// TIA Portal V20 export
FUNCTION "取芯伺服" : Void   // FC2, LAD
{ S7_Optimized_Access := 'TRUE' }
// stored: SetENOAutomatically false
BEGIN

REGION Network 1 (SCL)
   "取芯V90控制字".%X0 := "G2_下载".位9;
   "取芯V90控制字".%X1 := "G2_下载".位10;
   "取芯V90控制字".%X2 := "G2_下载".位11;
   "取芯V90控制字".%X3 := "G2_下载".位12;
   "取芯V90控制字".%X4 := "G2_下载".位13;
   "取芯V90控制字".%X5 := "G2_下载".位14;
   "取芯V90控制字".%X6 := "G2_下载".位15;
   "取芯V90控制字".%X7 := "G2_下载".位16;

   "取_回原模式" := "G2_下载".整型2;

   "取_绝对位置" := "G2_下载".浮点数6;
   "取_绝对速度" := "G2_下载".浮点数7;
   "取_相对位置" := "G2_下载".浮点数8;
   "取_相对位置" := "G2_下载".浮点数9;
   "取_点动速度" := "G2_下载".浮点数10;
END_REGION

REGION Network 2
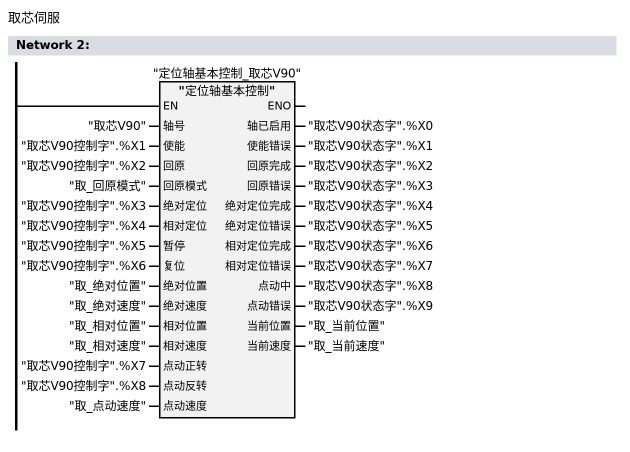
   RUNG wire#powerrail
      "定位轴基本控制_取芯V90"(轴号 := "取芯V90", 使能 := "取芯V90控制字".%X1, 回原 := "取芯V90控制字".%X2, 回原模式 := "取_回原模式", 绝对定位 := "取芯V90控制字".%X3, 相对定位 := "取芯V90控制字".%X4, 暂停 := "取芯V90控制字".%X5, 复位 := "取芯V90控制字".%X6, 绝对位置 := "取_绝对位置", 绝对速度 := "取_绝对速度", 相对位置 := "取_相对位置", 相对速度 := "取_相对速度", 点动正转 := "取芯V90控制字".%X7, 点动反转 := "取芯V90控制字".%X8, 点动速度 := "取_点动速度", 轴已启用 => "取芯V90状态字".%X0, 使能错误 => "取芯V90状态字".%X1, 回原完成 => "取芯V90状态字".%X2, 回原错误 => "取芯V90状态字".%X3, 绝对定位完成 => "取芯V90状态字".%X4, 绝对定位错误 => "取芯V90状态字".%X5, 相对定位完成 => "取芯V90状态字".%X6, 相对定位错误 => "取芯V90状态字".%X7, 点动中 => "取芯V90状态字".%X8, 点动错误 => "取芯V90状态字".%X9, 当前位置 => "取_当前位置", 当前速度 => "取_当前速度")
   END_RUNG
   // the same network as SCL:
   "定位轴基本控制_取芯V90"(轴号 := "取芯V90",   // "定位轴基本控制"
                   使能 := "取芯V90控制字".%X1,
                   回原 := "取芯V90控制字".%X2,
                   回原模式 := "取_回原模式",
                   绝对定位 := "取芯V90控制字".%X3,
                   相对定位 := "取芯V90控制字".%X4,
                   暂停 := "取芯V90控制字".%X5,
                   复位 := "取芯V90控制字".%X6,
                   绝对位置 := "取_绝对位置",
                   绝对速度 := "取_绝对速度",
                   相对位置 := "取_相对位置",
                   相对速度 := "取_相对速度",
                   点动正转 := "取芯V90控制字".%X7,
                   点动反转 := "取芯V90控制字".%X8,
                   点动速度 := "取_点动速度",
                   轴已启用 => "取芯V90状态字".%X0,
                   使能错误 => "取芯V90状态字".%X1,
                   回原完成 => "取芯V90状态字".%X2,
                   回原错误 => "取芯V90状态字".%X3,
                   绝对定位完成 => "取芯V90状态字".%X4,
                   绝对定位错误 => "取芯V90状态字".%X5,
                   相对定位完成 => "取芯V90状态字".%X6,
                   相对定位错误 => "取芯V90状态字".%X7,
                   点动中 => "取芯V90状态字".%X8,
                   点动错误 => "取芯V90状态字".%X9,
                   当前位置 => "取_当前位置",
                   当前速度 => "取_当前速度");
END_REGION

REGION Network 3 (SCL)
   "G2_上传".位11 := "取芯V90状态字".%X0;
   "G2_上传".位12 := "取芯V90状态字".%X1;
   "G2_上传".位13 := "取芯V90状态字".%X2;
   "G2_上传".位14 := "取芯V90状态字".%X3;
   "G2_上传".位15 := "取芯V90状态字".%X4;
   "G2_上传".位16 := "取芯V90状态字".%X5;
   "G2_上传".位17 := "取芯V90状态字".%X6;
   "G2_上传".位18 := "取芯V90状态字".%X7;
   "G2_上传".位19 := "取芯V90状态字".%X8;
   "G2_上传".位20 := "取芯V90状态字".%X9;

   "G2_上传".浮点数3 := LREAL_TO_REAL(IN := "取_当前位置");
   "G2_上传".浮点数4 := LREAL_TO_REAL(IN := "取_当前速度");
END_REGION
END_FUNCTION
